// TwinCAT 3 PLC project Untitled1
// ProgramVersion: 3.1.4024.0
// libraries:
//   Tc2_Standard, * (Beckhoff Automation GmbH)
//   Tc2_System, * (Beckhoff Automation GmbH)
//   Tc3_Module, * (Beckhoff Automation GmbH)
// project tree:
//   FB/ FB_ST10.TcPOU
//   / PlcTask.TcTTO (not stored)
//   POUs/ MAIN.TcPOU
// real-time tasks:
//   TASK PlcTask: cycle T#10ms, priority 20, ADS port 350

// ---- FB/FB_ST10.TcPOU
FUNCTION_BLOCK FB_ST10
VAR
	_camera : BOOL;
	_triger : BOOL;
	_description : STRING;
	_test : BOOL;
	_cameraProgram : UINT;
	_gitTest : BOOL;
	_git : INT;
END_VAR

METHOD PROTECTED _camera
VAR_INPUT
END_VAR
IF _camera THEN 
	_description:= 'On';
ELSE 
	_triger:= TRUE; 
END_IF
END_METHOD

METHOD _scanner : BOOL
VAR_INPUT
END_VAR
IF _triger THEN 
	_description:= 'Trger scanner';
END_IF
_gitTest:= TRUE;
END_METHOD

END_FUNCTION_BLOCK

// ---- POUs/MAIN.TcPOU
PROGRAM MAIN
VAR
END_VAR

END_PROGRAM
